FUNCTION_BLOCK FB_DiagnosisEtherCATSlaveWc1 IMPLEMENTS I_DiagnosisEtherCATSlave
VAR_INPUT
	sSlaveName					:STRING	:='NameNotSet';				//スレーブ名
END_VAR
VAR
	_bError						:BOOL;
	
	fbStateDiagnosis			:FB_StateDiagnosis;
	fbWcStateDiagnosis			:FB_WcStateDiagnosis;
END_VAR

(*エラー発生を出力*)
PROPERTY bError : BOOL
GET
bError:=_bError;
END_GET
END_PROPERTY

(*呼び出して診断実行*)
METHOD Execute
//診断用FBを呼び出し
fbStateDiagnosis(sSlaveName:=sSlaveName);
fbWcStateDiagnosis(sSlaveName:=sSlaveName);

_bError:=fbStateDiagnosis.bError OR fbWcStateDiagnosis.bError;
END_METHOD

END_FUNCTION_BLOCK

(* stored: Version 1.1.0.1
   POU FB_DiagnosisEtherCATSlaveWc1: Id {e5af8d40-9ba8-4884-bbf0-fd8f1590eb8a}, SpecialFunc None
   Property bError: Id {1aff0db5-352e-4661-a3e9-e533d01f3465}
   Get Get: Id {82095e75-b193-4035-bb84-01ec964d1d10}
   Method Execute: Id {0f30d909-8798-4d54-8e47-65e9a0221971} *)
